TYPE OutputBase_10CEE7DE :
STRUCT
END_STRUCT
END_TYPE

(* stored: Version 1.2.0.0, ProductVersion 3.1.4024.9
   DUT OutputBase_10CEE7DE: Id {9d02679b-624d-4923-9a72-5c5f805a9d76} *)
